// Mitsubishi GX Works2 project: Main_plc   PLC: FX3U/FX3UC

PROGRAM MAIN
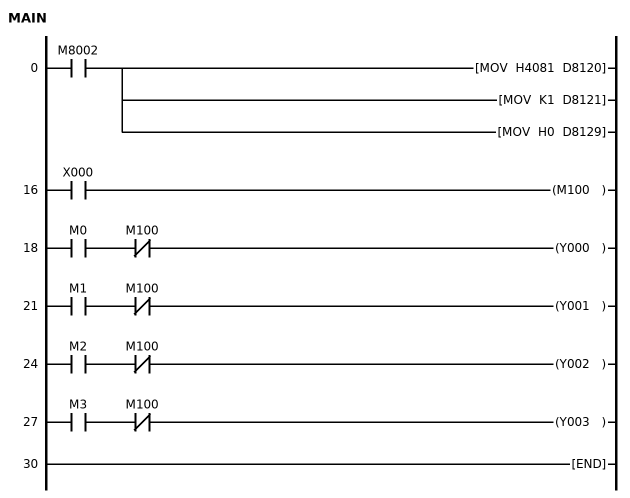
0     LD      M8002
      MOV     H4081 D8120
      MOV     K1 D8121
      MOV     H0 D8129
16    LD      X000
      OUT     M100
18    LD      M0
      ANI     M100
      OUT     Y000
21    LD      M1
      ANI     M100
      OUT     Y001
24    LD      M2
      ANI     M100
      OUT     Y002
27    LD      M3
      ANI     M100
      OUT     Y003
30    END
END_PROGRAM
